PROGRAM BH0MPL_LineBackground
VAR
END_VAR

MAIN.stLine_BH0MPL.fbLine(stLine:=MAIN.stLine_BH0MPL);
MAIN.stLine_BH0MPL.stStation_BH0MPL01.fbStation(
				stLine:=MAIN.stLine_BH0MPL,
				stStation:=MAIN.stLine_BH0MPL.stStation_BH0MPL01);

END_PROGRAM

(* stored: Version 1.1.0.1, ProductVersion 3.1.4024.15
   POU BH0MPL_LineBackground: Id {235f7efa-74f4-4f15-be11-c697478b11ac}, SpecialFunc None *)
